Staubli VAL3: _stopSimul.pgx

program _stopSimul()
  local string l_sEmpty
begin
  // reset the bit
  stopMove()
  // STOP SIMULATION
  logMsg("[KERNEL] SUPERVISOR:Cycle>Stop Simulation")
  // kill the task...
  taskKill("Simulation")
  taskKill("Action")
  watch(taskStatus("Simulation")==-1 and taskStatus("Action")==-1,1)
  //
  resetMotion()
  call OnEvent:OnCycleEvent(10)
end
